(* CODESYS project osmos_MXO_added.export

Project tree, tasks and I/O mapping:
  DUT/
    data type AI_Ctr
    data type AI_Par
    data type AO_Ctr
    data type AO_Par
    data type DI_Ctr
    data type DI_Par
    data type DO_Ctr
    data type DO_Par
    data type Motor_Ctr
    data type Motor_Data
    data type Motor_Par
    data type Valve_Ctr
    data type Valve_Data
    data type Valve_Par
  FB/
    CM/
      function block CM_AI [ST]
      function block CM_AO [ST]
      function block CM_DI [ST]
      function block CM_DO [ST]
      function block CM_Motor_dozz [ST]
      function block CM_Valve_dozz [ST]
    function block CLK_1_sec [ST]
    function block _USR_CTU [ST]
  Popup/
    visualisation popup_AI
    visualisation popup_AO
    visualisation popup_DO
    visualisation popup_Motor
    visualisation popup_Sensor
    visualisation popup_Valve
*)

// DUT/AI_Ctr
TYPE AI_Ctr :
STRUCT
	ManMode:		BOOL := FALSE; //False - Auto, True - Manual
	ManValue:		REAL; 
END_STRUCT
END_TYPE

// DUT/AI_Par
TYPE AI_Par :
STRUCT
	Raw_MIN:		REAL := 0;
	Raw_MAX:		REAL := 100;
	Eng_MIN:		REAL := 0;
	Eng_MAX:		REAL := 100;
	Filter_Constant:REAL;// From 0 to 1
	Filter_Time:	UINT;//Time for filter in seconds	
END_STRUCT
END_TYPE

// DUT/AO_Ctr
TYPE AO_Ctr :
STRUCT
	ManMode:		BOOL := FALSE; //False - Auto, True - Manual
	ManValue:		REAL; 
END_STRUCT
END_TYPE

// DUT/AO_Par
TYPE AO_Par :
STRUCT	
	Eng_MIN:		REAL := 0;
	Eng_MAX:		REAL := 100;
	Raw_MIN:		REAL := 0;
	Raw_MAX:		REAL :=1000;
END_STRUCT
END_TYPE

// DUT/DI_Ctr
TYPE DI_Ctr :
STRUCT
	ManMode:		BOOL := FALSE; //False - Auto, True - Manual
	ManAct:			BOOL; 
END_STRUCT
END_TYPE

// DUT/DI_Par
TYPE DI_Par :
STRUCT
	Debounce_On:	UINT := 100; //Delay in milliseconds
	Debounce_Off:	UINT := 100; //Delay in milliseconds
END_STRUCT
END_TYPE

// DUT/DO_Ctr
TYPE DO_Ctr :
STRUCT
	ManMode:		BOOL := FALSE; //False - Auto, True - Manual
	ManAct:			BOOL; 
END_STRUCT
END_TYPE

// DUT/DO_Par
TYPE DO_Par :
STRUCT
	Debounce_On:	UINT; //Delay in milliseconds
	Debounce_Off:	UINT; //Delay in milliseconds
END_STRUCT
END_TYPE

// DUT/Motor_Ctr
TYPE Motor_Ctr :
STRUCT
	ManMode:		BOOL := FALSE; //False - Auto, True - Manual
	ManAct:			BOOL;
	AlmSuppress:	BOOL; 
END_STRUCT
END_TYPE

// DUT/Motor_Data
TYPE Motor_Data :
STRUCT
	xActivate:		BOOL;
	xFault:			BOOL;
	xOut:			BOOL;
	dwColor:		DWORD;
END_STRUCT
END_TYPE

// DUT/Motor_Par
TYPE Motor_Par :
STRUCT
	On_Delay:		UINT := 0; //all delays are set in seconds only
	Off_Delay:		UINT := 0;
	ActFlt_Delay:	UINT := 5;
	DeactFlt_Delay:	UINT := 5;
END_STRUCT
END_TYPE

// DUT/Valve_Ctr
TYPE Valve_Ctr :
STRUCT
	ManMode:		BOOL := FALSE; //False - Auto, True - Manual
	ManAct:			BOOL;
	ManActUS:		BOOL;
	ManActLS:		BOOL;
	AlmSuppress:	BOOL; 
END_STRUCT
END_TYPE

// DUT/Valve_Data
TYPE Valve_Data :
STRUCT
	xActivate:		BOOL;
	xActUpSeat:		BOOL;
	xActLowSeat:	BOOL;
	xFault:			BOOL;
	xOut:			BOOL;
	dwColor:		DWORD;
END_STRUCT
END_TYPE

// DUT/Valve_Par
TYPE Valve_Par :
STRUCT
	On_Delay:		UINT := 0; //all delays are set in seconds only
	Off_Delay:		UINT := 0;
	ActFlt_Delay:	UINT := 8;
	DeactFlt_Delay:	UINT := 8;	
END_STRUCT
END_TYPE

// FB/CLK_1_sec
FUNCTION_BLOCK CLK_1_sec
VAR_INPUT
	EN:		BOOL;
	PT:		TIME := T#1S;
END_VAR
VAR_OUTPUT
	Q:		BOOL;
END_VAR
VAR
	M:		BOOL;
	t_last:	TIME;
	tm:		TIME;
END_VAR

// This block is used for making blink-signal in a certain time with duration 1 cycle

tm := TIME();
// R_TRIG for initialization, to enable Q, when start
IF EN AND NOT M THEN
	t_last := tm - PT;  
END_IF
M := EN;

Q := tm - t_last > PT;
IF Q THEN
	t_last := tm;
END_IF

END_FUNCTION_BLOCK

// FB/_USR_CTU
FUNCTION_BLOCK _USR_CTU
VAR_INPUT
	EN:		BOOL;
	PV:		UINT;// Preset value
	CU:		BOOL;// Count input
END_VAR
VAR_OUTPUT
	Q:		BOOL;// Output
	CV:		UINT;// Current value
END_VAR
VAR	
END_VAR

// user counter up is made, to be used in ST (because in standart variant no EN/ENO)
IF NOT EN THEN
	Q := FALSE;
	CV := 0;
	RETURN;
ELSE
	IF NOT Q AND CU THEN
		CV := CV + 1;// Increase value by 1 while EN is TRUE and NOT Q
	END_IF
END_IF
Q := CV >= PV;

END_FUNCTION_BLOCK

// FB/CM/CM_AI
FUNCTION_BLOCK CM_AI
VAR_INPUT
	Name:			STRING;
	rIn:			REAL;
	Par:			AI_Par;
END_VAR
VAR_IN_OUT
	Ctrl:			AI_Ctr;
END_VAR
VAR_OUTPUT
	rOut:			REAL;
END_VAR
VAR
	xManModeMem:	BOOL;
	rOutMem:		REAL;
END_VAR
VAR_TEMP
	rOutTmp:		REAL;
END_VAR

// Scale 4..20 mA to 0..100% (for example)
rOutTmp := SCALE_R(
		IN:= rIn, 
		IN_LO:= Par.Raw_MIN, 
		IN_HI:= Par.Raw_MAX, 
		OUT_LO:= Par.Eng_MIN, 
		OUT_HI:= Par.Eng_MAX);
		
// Auto-Manual mode		
IF Ctrl.ManMode THEN
	IF NOT xManModeMem THEN // R_TRIG
		Ctrl.ManValue := rOutTmp;
	END_IF
	rOutTmp := Ctrl.ManValue; // Assign Man value in Engineering unit to Out (after scale)
END_IF
xManModeMem := Ctrl.ManMode; // Memory bit for R_TRIG Man mode

// Filter 
IF PLC_PRG.xFirstScan THEN//Initialization
	rOutMem := 0;
END_IF

IF Par.Filter_Constant < 1 AND Par.Filter_Constant > 0 AND NOT Ctrl.ManMode THEN
	rOutTmp := Par.Filter_Constant * rOutMem + (1 - Par.Filter_Constant) * rOutTmp;
END_IF

rOut := rOutMem := rOutTmp;

END_FUNCTION_BLOCK

// FB/CM/CM_AO
FUNCTION_BLOCK CM_AO
VAR_INPUT
	Name:			STRING;
	rIn:			REAL;
	Par:			AO_Par;
END_VAR
VAR_IN_OUT
	Ctrl:			AO_Ctr;
END_VAR
VAR_OUTPUT
	rOut:			REAL;
	rOutVisu:		REAL;
END_VAR
VAR
	xManModeMem:	BOOL;	
END_VAR
VAR_TEMP
	rInTmp: 		REAL;		
END_VAR

rInTmp := rIn;

// Auto-Manual mode	
IF Ctrl.ManMode THEN
	IF NOT xManModeMem THEN // R_TRIG
		Ctrl.ManValue := rInTmp;
	END_IF
	rInTmp := Ctrl.ManValue; // Assign Man value in Engineering unit to In before scale
END_IF
xManModeMem := Ctrl.ManMode; //Memory bit for R_TRIG Man mode
rOutVisu := rInTmp;
// Scale from Engineering unit to Raw value (for example: 0..100% => 4..20 mA)
rOut := SCALE_R(
		IN:= rInTmp, 
		IN_LO:= Par.Eng_MIN, 
		IN_HI:= Par.Eng_MAX, 
		OUT_LO:= Par.Raw_MIN, 
		OUT_HI:= Par.Raw_MAX);

END_FUNCTION_BLOCK

// FB/CM/CM_DI
FUNCTION_BLOCK CM_DI
VAR_INPUT
	Name:		STRING;
	xIn:		BOOL;
	Par:		DI_par;
END_VAR
VAR_IN_OUT
	Ctrl:		DI_Ctr;
END_VAR
VAR_OUTPUT
	xOut:		BOOL;
END_VAR
VAR
	xM:			BOOL;
	xManModeMem:BOOL;
	tStart:		TIME;	
END_VAR
VAR_TEMP
	tmpDebounceON:	TIME;
	tmpDebounceOFF:	TIME;
END_VAR

xOut := xIn;// Activation without filters when Parameters = 0

// Delay to activate output
IF Par.Debounce_On >0 THEN 
	tmpDebounceON := UINT_TO_TIME(Par.Debounce_On);
	IF xIn AND NOT xM THEN// R_TRIG
		tStart := TIME();
	END_IF
	xOut := xIn AND ((TIME() - tStart) > tmpDebounceON);		
END_IF

// Delay to deactivate output
IF Par.Debounce_Off >0 THEN
	tmpDebounceOFF := UINT_TO_TIME(Par.Debounce_Off);
	IF xM AND NOT xIn THEN// F_TRIG
		tStart := TIME();
	END_IF
	IF NOT xIn AND ((TIME() - tStart) < tmpDebounceOFF) THEN
		xOut := TRUE;
	END_IF		
END_IF

IF Ctrl.ManMode THEN
	IF NOT xManModeMem THEN
		Ctrl.ManAct := xOut;
	END_IF
	xOut := Ctrl.ManAct;
END_IF

xM := xIn;
xManModeMem := Ctrl.ManMode;

END_FUNCTION_BLOCK

// FB/CM/CM_DO
FUNCTION_BLOCK CM_DO
VAR_INPUT
	Name:		STRING;
	xIn:		BOOL;
	Par:		DO_par;
END_VAR
VAR_IN_OUT
	Ctrl:		DO_Ctr;
END_VAR
VAR_OUTPUT
	xOut:		BOOL;
END_VAR
VAR
	xM:			BOOL;
	xManModeMem:BOOL;
	tStart:		TIME;	
END_VAR
VAR_TEMP
	tmpDebounceON:	TIME;
	tmpDebounceOFF:	TIME;
END_VAR

xOut := xIn;// Activation without filters when Parameters = 0

// Delay to activate output
IF Par.Debounce_On >0 THEN 
	tmpDebounceON := UINT_TO_TIME(Par.Debounce_On);
	IF xIn AND NOT xM THEN// R_TRIG
		tStart := TIME();
	END_IF
	xOut := xIn AND ((TIME() - tStart) > tmpDebounceON);		
END_IF

// Delay to deactivate output
IF Par.Debounce_Off >0 THEN
	tmpDebounceOFF := UINT_TO_TIME(Par.Debounce_Off);
	IF xM AND NOT xIn THEN// F_TRIG
		tStart := TIME();
	END_IF
	IF NOT xIn AND ((TIME() - tStart) < tmpDebounceOFF) THEN
		xOut := TRUE;
	END_IF		
END_IF

IF Ctrl.ManMode THEN
	IF NOT xManModeMem THEN
		Ctrl.ManAct := xOut;
	END_IF
	xOut := Ctrl.ManAct;
END_IF

xM := xIn;
xManModeMem := Ctrl.ManMode;

END_FUNCTION_BLOCK

// FB/CM/CM_Motor_dozz
FUNCTION_BLOCK CM_Motor_dozz
VAR_INPUT
	Name:			STRING;
	Config:			BYTE;	
	FB:				BOOL;
	Rst:			BOOL;
	Motor_Par:		Motor_Par;
END_VAR
VAR_IN_OUT
	Act:			BOOL;
	Motor_Ctr:		Motor_Ctr;
END_VAR
VAR_OUTPUT
	Q:				BOOL;
	Flt:			BOOL;
END_VAR
VAR
	D_F_CTU:		_USR_CTU;
	A_F_CTU:		_USR_CTU;
	D_D_CTU:		_USR_CTU;
	A_D_CTU:		_USR_CTU;
	xAct:			BOOL;	
	xDeAct:			BOOL;
	xActDlyDone:	BOOL;
	xDeActDlyDone:	BOOL;
	Act_temp_old:	BOOL;
	ManModeMem:		BOOL;
	xGlobalAlmSupMem:	BOOL;
	dwColor:		DWORD;	
END_VAR
VAR_TEMP
	Act_temp:		BOOL;
	FB_En:			BOOL;
	RstIn_En:		BOOL;
END_VAR

Q := FALSE; 

// Read config
FB_En 		:= Config.0;
RstIn_En 	:= Config.1;

// Read parameters
A_F_CTU(PV := Motor_Par.ActFlt_Delay, CU := PLC_PRG.xCLK_1_sec);// parameters for act fault
D_F_CTU(PV := Motor_Par.DeactFlt_Delay, CU := PLC_PRG.xCLK_1_sec);// parameters for deact fault
A_D_CTU(PV := Motor_Par.On_Delay, CU:= PLC_PRG.xCLK_1_sec);// parameters for act delay
D_D_CTU(PV := Motor_Par.Off_Delay, CU:= PLC_PRG.xCLK_1_sec);// parameters for deact delay

// Reset input
IF RstIn_En THEN
	Act_temp := Act;	// Assign input to to internal variable
	Act := FALSE;
END_IF

// Auto/Man mode
IF Motor_Ctr.ManMode THEN
	IF NOT ManModeMem THEN // Detect R_trig
		Motor_Ctr.ManAct := Act_temp;		
	END_IF
	Act_temp := Motor_Ctr.ManAct;	
END_IF
ManModeMem := Motor_Ctr.ManMode;

// Activations
// Detect F_trig and R_trig activation, to SET/RESET timers
IF Act_temp AND NOT Act_temp_old THEN// R_trig activation
	xAct := TRUE;// set value on activation	
	xDeAct := FALSE;
	xActDlyDone := FALSE;
	IF NOT xDeActDlyDone THEN
		xActDlyDone := TRUE;// disable Act delay timer if DeAct delay timer is not done (Motor is activated yet)
	END_IF
	D_D_CTU.EN := FALSE;
END_IF
IF Act_temp_old AND NOT Act_temp THEN// F_trig activation
	xDeAct := TRUE;
	xAct :=FALSE;
	xDeActDlyDone := FALSE;
	IF NOT xActDlyDone THEN
		xDeActDlyDone := TRUE; // disable DeAct delay timer if Act delay timer is not done (Motor is not activated yet)
	END_IF
	A_D_CTU.EN := FALSE;
END_IF

// Activation delay
IF xAct THEN
	IF A_D_CTU.PV > 0 AND NOT xActDlyDone THEN
		A_D_CTU.EN := TRUE;//start timer 
		IF A_D_CTU.Q THEN
			xActDlyDone :=TRUE;
			A_D_CTU.EN := FALSE;
		END_IF	
	ELSE
		Q := Act_temp;
	END_IF	
END_IF
	
// Deactivation delay
IF xDeAct THEN
	IF D_D_CTU.PV > 0 AND NOT xDeActDlyDone THEN
		D_D_CTU.EN := TRUE;//Start timer
		Q := TRUE; 
		IF 	D_D_CTU.Q THEN
			xDeActDlyDone := TRUE;
			D_D_CTU.EN := FALSE;			
		END_IF
	ELSE
		Q := Act_temp;
	END_IF
END_IF


 //Activating fault timers, when Feedback is used	
IF FB_En THEN
	// Act_fault delay
	IF xAct AND Q AND NOT FB THEN
		A_F_CTU.EN :=TRUE;// Start timer 
		IF A_F_CTU.Q THEN 
			Flt := TRUE;
		END_IF
	ELSE
		A_F_CTU.EN := FALSE;
	END_IF
	// Deact fault delay
	IF xDeAct AND FB AND NOT Q THEN
		D_F_CTU.EN :=TRUE;// Start timer 
		IF D_F_CTU.Q THEN
			Flt := TRUE;
		END_IF
	ELSE
		D_F_CTU.EN :=FALSE;
	END_IF
END_IF

// Global fault reset handling
IF PLC_PRG.xGlobalAlmSup AND NOT xGlobalAlmSupMem THEN
	Motor_Ctr.AlmSuppress := TRUE;
END_IF
IF xGlobalAlmSupMem  AND NOT PLC_PRG.xGlobalAlmSup THEN
	Motor_Ctr.AlmSuppress := FALSE;
END_IF
xGlobalAlmSupMem := PLC_PRG.xGlobalAlmSup;

// Fault reset
IF Motor_Ctr.AlmSuppress OR Rst THEN
	Flt := FALSE;
END_IF

// Colors
dwColor := Const.Color_Def;

IF Q THEN
	dwColor := Const.Color_Green;
END_IF

IF Flt THEN
	dwColor := Const.Color_Fault;
END_IF

Act_temp_old := Act_temp;

END_FUNCTION_BLOCK

// FB/CM/CM_Valve_dozz
FUNCTION_BLOCK CM_Valve_dozz
VAR_INPUT
	Name:			STRING;
	Config:			BYTE;	
	FB:				BOOL;
	Rst:			BOOL;
	Act_UpperSeat:	BOOL;
	Act_LowerSeat:	BOOL;
	Valve_Par:		Valve_Par;
END_VAR
VAR_IN_OUT
	Act:			BOOL;

	Valve_Ctr:		Valve_Ctr;
END_VAR
VAR_OUTPUT
	Q:				BOOL;
	Q_UpperSeat:	BOOL;
	Q_LowerSeat:	BOOL;
	Flt:			BOOL;
	dwColor:		DWORD;
END_VAR
VAR
	D_F_CTU:		_USR_CTU;
	A_F_CTU:		_USR_CTU;
	D_D_CTU:		_USR_CTU;
	A_D_CTU:		_USR_CTU;
	xAct:			BOOL;	
	xDeAct:			BOOL;
	xActDlyDone:	BOOL;
	xDeActDlyDone:	BOOL;
	Act_temp_old:	BOOL;
	ManModeMem:		BOOL;
END_VAR
VAR_TEMP
	Act_temp:		BOOL;
	Act_US_temp:	BOOL;
	Act_LS_temp:	BOOL;
	FB_En:			BOOL;
	FB_temp:		BOOL;
	RstIn_En:		BOOL;
END_VAR

Q := Q_UpperSeat := Q_LowerSeat := FALSE; 
Act_temp := Act;// Assighn input to to internal variable

// Read config
FB_En 		:= Config.0;
RstIn_En 	:= Config.1;

FB_temp := FB;
IF Config.3 THEN // deact FB
	FB_temp := NOT FB;
END_IF

// Read parameters
A_F_CTU(PV := Valve_Par.ActFlt_Delay, CU := PLC_PRG.xCLK_1_sec);// parameters for act fault
D_F_CTU(PV := Valve_Par.DeactFlt_Delay, CU := PLC_PRG.xCLK_1_sec);// parameters for deact fault
A_D_CTU(PV := Valve_Par.On_Delay, CU:= PLC_PRG.xCLK_1_sec);// parameters for act delay
D_D_CTU(PV := Valve_Par.Off_Delay, CU:= PLC_PRG.xCLK_1_sec);// parameters for deact delay

// Seat temp act
Act_US_temp := Act_UpperSeat;
Act_LS_temp := Act_LowerSeat;

// Auto/Man mode
IF Valve_Ctr.ManMode THEN
	IF NOT ManModeMem THEN // Detect R_trig
		Valve_Ctr.ManAct := Act_temp;
		Valve_Ctr.ManActUS := Act_US_temp;
		Valve_Ctr.ManActLS := Act_LS_temp;
	END_IF
	Act_temp := Valve_Ctr.ManAct;
	Act_US_temp := Valve_Ctr.ManActUS;
	Act_LS_temp := Valve_Ctr.ManActLS;
END_IF
ManModeMem := Valve_Ctr.ManMode;

// Activations
// Detect F_trig and R_trig activation, to SET/RESET timers
IF Act_temp AND NOT Act_temp_old THEN// R_trig activation
	xAct := TRUE;// set value on activation	
	xDeAct := FALSE;
	xActDlyDone := FALSE;
	IF NOT xDeActDlyDone THEN
		xActDlyDone := TRUE;// disable Act delay timer if DeAct delay timer is not done (valve is activated yet)
	END_IF
	D_D_CTU.EN := FALSE;
END_IF
IF Act_temp_old AND NOT Act_temp THEN// F_trig activation
	xDeAct := TRUE;
	xAct :=FALSE;
	xDeActDlyDone := FALSE;
	IF NOT xActDlyDone THEN
		xDeActDlyDone := TRUE; // disable DeAct delay timer if Act delay timer is not done (valve is not activated yet)
	END_IF
	A_D_CTU.EN := FALSE;
END_IF

// Activation delay
IF xAct THEN
	IF A_D_CTU.PV > 0 AND NOT xActDlyDone THEN
		A_D_CTU.EN := TRUE;//start timer 
		IF A_D_CTU.Q THEN
			xActDlyDone :=TRUE;
			A_D_CTU.EN := FALSE;
		END_IF	
	ELSE
		Q := Act_temp;
	END_IF	
END_IF
	
// Deactivation delay
IF xDeAct THEN
	IF D_D_CTU.PV > 0 AND NOT xDeActDlyDone THEN
		D_D_CTU.EN := TRUE;//Start timer
		Q := TRUE; 
		IF 	D_D_CTU.Q THEN
			xDeActDlyDone := TRUE;
			D_D_CTU.EN := FALSE;			
		END_IF
	ELSE
		Q := Act_temp;
	END_IF
END_IF


 //Activating fault timers, when Feedback is used	
IF FB_En THEN
	// Act_fault delay
	IF xAct AND Q AND NOT FB_temp THEN
		A_F_CTU.EN :=TRUE;// Start timer 
		IF A_F_CTU.Q THEN 
			Flt := TRUE;
		END_IF
	ELSE
		A_F_CTU.EN := FALSE;
	END_IF
	// Deact fault delay
	IF xDeAct AND FB_temp AND NOT Q THEN
		D_F_CTU.EN :=TRUE;// Start timer 
		IF D_F_CTU.Q THEN
			Flt := TRUE;
		END_IF
	ELSE
		D_F_CTU.EN :=FALSE;
	END_IF
END_IF

// Global fault reset
IF PLC_PRG.xGlobalAlmSup THEN
	Valve_Ctr.AlmSuppress := TRUE;
END_IF

// Fault reset
IF Valve_Ctr.AlmSuppress OR Rst THEN
	Flt := FALSE;
END_IF

// Seat activation
IF Config.2 THEN // Mixproof valve
	Q_UpperSeat := Act_US_temp;
	Q_LowerSeat := Act_LS_temp;
END_IF

// Colors
dwColor := Const.Color_Def;

IF Q THEN
	dwColor := Const.Color_Green;
END_IF

IF Flt THEN
	dwColor := Const.Color_Fault;
END_IF

Act_temp_old := Act_temp;

END_FUNCTION_BLOCK

// Popup/popup_AI
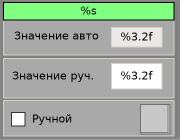
VISUALIZATION popup_AI  // 180x140
VAR_INPUT
	AICfg: 	POINTER TO CM_AI;
	AICtrl:	POINTER TO AI_Ctr;
END_VAR
    Rectangle (0,0 180x138)
        OnMouseClick: execute { SensorVis:=2; }
    Rectangle (3,2 171x53)
    Rectangle (3,2 171x18), "%s", text variable: AICfg^.Name
    Rectangle (3,100 171x36)
    Button (140,104 30x30), image: ImagePool.exit
        OnMouseClick:  Dialog=popup_AI, Result=OK, NumpadKeypadSet=True
    Rectangle (3,58 171x40)
    Label (9,61 95x30), "Значение руч."
    Checkbox (9,107 110x24), "Ручной", variable: AICtrl^.ManMode
    Textfield (111,63 51x26), "%3.2f", text variable: AICtrl^.ManValue, input disabled if: not AICtrl^.ManMode
        OnMouseClick: write the text variable via VisuDialogs.Numpad, min 0, max 100
    Label (11,21 95x30), "Значение авто"
    Textfield (111,27 51x20), "%3.2f", text variable: AICfg^.rOut
    hotkey  Id=481037385728, Key=KeyDown=True, KeyName=ESCAPE, VisuElemId=31
    hotkey  Id=481038434304, Key=KeyName=ESCAPE, VisuElemId=31
END_VISUALIZATION

// Popup/popup_AO
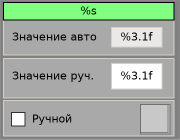
VISUALIZATION popup_AO  // 180x140
VAR_INPUT
	AOCfg: 	POINTER TO CM_AO;
	AOCtrl:	POINTER TO AO_Ctr;
END_VAR
    Rectangle (0,0 180x138)
        OnMouseClick: execute { SensorVis:=2; }
    Rectangle (3,2 171x53)
    Rectangle (3,2 171x18), "%s", text variable: AOCfg^.Name
    Rectangle (3,100 171x36)
    Button (140,104 30x30), image: ImagePool.exit
        OnMouseClick:  Dialog=popup_AO, Result=OK, NumpadKeypadSet=True
    Rectangle (3,58 171x40)
    Label (9,61 95x30), "Значение руч."
    Checkbox (9,107 110x24), "Ручной", variable: AOCtrl^.ManMode
    Textfield (111,63 51x26), "%3.1f", text variable: AOCtrl^.ManValue, input disabled if: not AOCtrl^.ManMode
        OnMouseClick: write the text variable via VisuDialogs.Numpad, min 0, max 100
    Label (9,22 95x30), "Значение авто"
    Textfield (111,27 51x20), "%3.1f", text variable: AOCfg^.rIn
    hotkey  Id=481037385728, Key=KeyDown=True, KeyName=ESCAPE, VisuElemId=31
    hotkey  Id=481038434304, Key=KeyName=ESCAPE, VisuElemId=31
END_VISUALIZATION

// Popup/popup_DO
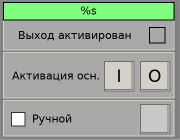
VISUALIZATION popup_DO  // 180x140
VAR_INPUT
	QCfg: 	POINTER TO CM_DO;
	QCtrl:	POINTER TO DO_Ctr;
END_VAR
    Rectangle (0,0 180x138)
        OnMouseClick: execute { SensorVis:=2; }
    Rectangle (3,2 171x48)
    Rectangle (3,2 171x18), "%s", text variable: QCfg^.Name
    Rectangle (3,100 171x36)
    Button (140,104 30x30), image: ImagePool.exit
        OnMouseClick:  Dialog=popup_DO, Result=OK, NumpadKeypadSet=True
    Rectangle (3,52 171x46)
    Label (9,61 95x30), "Активация осн."
    Rectangle (149,27 16x16), colour toggle: QCfg^.xOut
    Label (12,25 126x21), "Выход активирован"
    Checkbox (9,107 110x24), "Ручной", variable: QCtrl^.ManMode
    Button (104,61 30x30), "I", colour toggle: QCfg^.xOut, input disabled if: not QCtrl^.ManMode
        OnMouseClick: execute { QCtrl^.ManAct := TRUE; }
    Button (140,61 30x30), "O", colour toggle: not QCfg^.xOut, input disabled if: not QCtrl^.ManMode
        OnMouseClick: execute { QCtrl^.ManAct := FALSE; }
    hotkey  Id=481037385728, Key=KeyDown=True, KeyName=ESCAPE, VisuElemId=31
    hotkey  Id=481038434304, Key=KeyName=ESCAPE, VisuElemId=31
END_VISUALIZATION

// Popup/popup_Motor
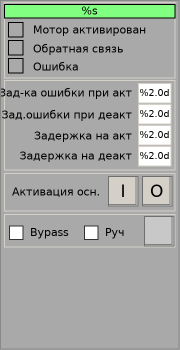
VISUALIZATION popup_Motor  // 180x350
//{attribute 'var_in_out_as_pointer'}
VAR_INPUT 
	M_Cfg: 	POINTER TO CM_Motor_dozz;
	M_Cmd:	POINTER TO Motor_Ctr;
	M_Par:	POINTER TO Motor_Par;
END_VAR
    Rectangle (4,80 171x90)
    Rectangle (4,2 171x76)
    Rectangle (4,4 171x14), "%s", text variable: M_Cfg^.Name
    Rectangle (4,214 171x33)
    Textfield (138,83 33x20), "%2.0d", text variable: M_Par^.ActFlt_Delay
        OnMouseClick: write the text variable via VisuDialogs.Numpad, min 0, max 99
    Label (6,78 129x30), "Зад-ка ошибки при акт"
    Textfield (138,104 33x20), "%2.0d", text variable: M_Par^.DeactFlt_Delay
        OnMouseClick: write the text variable via VisuDialogs.Numpad, min 0, max 99
    Label (6,100 129x30), "Зад.ошибки при деакт"
    Textfield (138,125 33x20), "%2.0d", text variable: M_Par^.On_Delay
        OnMouseClick: write the text variable via VisuDialogs.Numpad, min 0, max 30
    Label (7,121 128x30), "Задержка на акт"
    Textfield (138,146 33x20), "%2.0d", text variable: M_Par^.Off_Delay
        OnMouseClick: write the text variable via VisuDialogs.Numpad, min 0, max 30
    Label (7,141 128x30), "Задержка на деакт"
    Rectangle (4,173 171x38)
    Button (108,176 30x30), "I", colour toggle: M_Cfg^.Q, input disabled if: not M_Cmd^.ManMode
        OnMouseClick: execute { M_Cmd^.ManAct := TRUE; }
    Button (142,176 30x30), "O", colour toggle: not M_Cfg^.Q, input disabled if: not M_Cmd^.ManMode
        OnMouseClick: execute { M_Cmd^.ManAct := FALSE; }
    Label (9,177 95x30), "Активация осн."
    Checkbox (7,219 75x27), "Bypass", variable: M_Cmd^.AlmSuppress
    Checkbox (82,219 56x27), "Руч", variable: M_Cmd^.ManMode
    Button (144,216 30x30), image: ImagePool.exit
        OnMouseClick:  Dialog=popup_Motor, Result=OK, NumpadKeypadSet=True
    Label (30,21 126x18), "Мотор активирован"
    Rectangle (8,22 15x15), colour toggle: M_Cfg^.Q
    Rectangle (8,40 15x15), colour toggle: M_Cfg^.FB
    Label (30,40 126x18), "Обратная связь"
    Rectangle (8,58 15x15), colour toggle: M_Cfg^.Flt
    Label (30,58 57x18), "Ошибка"
END_VISUALIZATION

// Popup/popup_Sensor
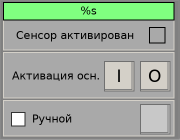
VISUALIZATION popup_Sensor  // 180x140
VAR_INPUT
	SCfg: 	POINTER TO CM_DI;
	SCtrl:	POINTER TO DI_Ctr;
END_VAR
    Rectangle (0,0 180x138)
        OnMouseClick: execute { SensorVis:=2; }
    Rectangle (3,2 171x48)
    Rectangle (3,2 171x18), "%s", text variable: SCfg^.Name
    Rectangle (3,100 171x36)
    Button (140,104 30x30), image: ImagePool.exit
        OnMouseClick:  Dialog=popup_Sensor, Result=OK, NumpadKeypadSet=True
    Rectangle (3,52 171x46)
    Label (9,61 95x30), "Активация осн."
    Rectangle (149,27 16x16), colour toggle: SCfg^.xOut
    Label (12,25 126x21), "Сенсор активирован"
    Checkbox (9,107 110x24), "Ручной", variable: SCtrl^.ManMode
    Button (104,61 30x30), "I", colour toggle: SCfg^.xOut, input disabled if: not SCtrl^.ManMode
        OnMouseClick: execute { SCtrl^.ManAct := TRUE; }
    Button (140,61 30x30), "O", colour toggle: not SCfg^.xOut, input disabled if: not SCtrl^.ManMode
        OnMouseClick: execute { SCtrl^.ManAct := FALSE; }
    hotkey  Id=481037385728, Key=KeyDown=True, KeyName=ESCAPE, VisuElemId=31
    hotkey  Id=481038434304, Key=KeyName=ESCAPE, VisuElemId=31
END_VISUALIZATION

// Popup/popup_Valve
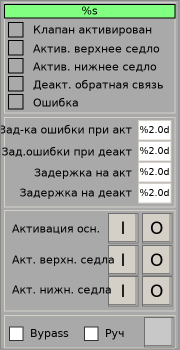
VISUALIZATION popup_Valve  // 180x350
//{attribute 'var_in_out_as_pointer'}
VAR_INPUT 
	V_Cfg: 	POINTER TO CM_Valve_dozz;
	V_Cmd:	POINTER TO Valve_Ctr;
	V_Par:	POINTER TO Valve_Par;
END_VAR
    Rectangle (4,117 171x90)
    Rectangle (4,2 171x111)
    Rectangle (4,4 171x14), "%s", text variable: V_Cfg^.Name
    Rectangle (4,315 171x33)
    Textfield (138,120 33x20), "%2.0d", text variable: V_Par^.ActFlt_Delay
        OnMouseClick: write the text variable via VisuDialogs.Numpad, min 0, max 99
    Label (6,115 129x30), "Зад-ка ошибки при акт"
    Textfield (138,141 33x20), "%2.0d", text variable: V_Par^.DeactFlt_Delay
        OnMouseClick: write the text variable via VisuDialogs.Numpad, min 0, max 99
    Label (6,137 129x30), "Зад.ошибки при деакт"
    Textfield (138,162 33x20), "%2.0d", text variable: V_Par^.On_Delay
        OnMouseClick: write the text variable via VisuDialogs.Numpad, min 0, max 30
    Label (7,158 128x30), "Задержка на акт"
    Textfield (138,183 33x20), "%2.0d", text variable: V_Par^.Off_Delay
        OnMouseClick: write the text variable via VisuDialogs.Numpad, min 0, max 30
    Label (7,178 128x30), "Задержка на деакт"
    Rectangle (4,210 171x101)
    Button (108,213 30x30), "I", colour toggle: V_Cfg^.Q, input disabled if: not V_Cmd^.ManMode
        OnMouseClick: execute { V_Cmd^.ManAct := TRUE; }
    Button (142,213 30x30), "O", colour toggle: not V_Cfg^.Q, input disabled if: not V_Cmd^.ManMode
        OnMouseClick: execute { V_Cmd^.ManAct := FALSE; }
    Button (108,245 30x30), "I", colour toggle: V_Cfg^.Q_UpperSeat, input disabled if: not V_Cmd^.ManMode
        OnMouseClick: execute { V_Cmd^.ManActUS := TRUE; }
    Button (142,245 30x30), "O", colour toggle: not V_Cfg^.Q_UpperSeat, input disabled if: not V_Cmd^.ManMode
        OnMouseClick: execute { V_Cmd^.ManActUS := FALSE; }
    Button (108,276 30x30), "I", colour toggle: V_Cfg^.Q_LowerSeat, input disabled if: not V_Cmd^.ManMode
        OnMouseClick: execute { V_Cmd^.ManActLS := TRUE; }
    Button (142,276 30x30), "O", colour toggle: not V_Cfg^.Q_LowerSeat, input disabled if: not V_Cmd^.ManMode
        OnMouseClick: execute { V_Cmd^.ManActLS := FALSE; }
    Label (9,214 95x30), "Активация осн."
    Label (9,245 103x30), "Акт. верхн. седла"
    Label (9,275 103x30), "Акт. нижн. седла"
    Checkbox (7,320 75x27), "Bypass", variable: V_Cmd^.AlmSuppress
    Checkbox (82,320 56x27), "Руч", variable: V_Cmd^.ManMode
    Button (144,317 30x30), image: ImagePool.exit
        OnMouseClick:  Dialog=popup_Valve, Result=OK, NumpadKeypadSet=True
    Label (30,21 126x18), "Клапан активирован"
    Rectangle (8,22 15x15), colour toggle: V_Cfg^.Q
    Rectangle (8,40 15x15), colour toggle: V_Cfg^.Q_UpperSeat
    Label (30,40 126x18), "Актив. верхнее седло"
    Rectangle (8,58 15x15), colour toggle: V_Cfg^.Q_LowerSeat
    Label (30,58 126x18), "Актив. нижнее седло"
    Rectangle (8,76 15x15), colour toggle: V_Cfg^.FB
    Label (30,76 126x18), "Деакт. обратная связь"
    Rectangle (8,94 15x15), colour toggle: V_Cfg^.Flt
    Label (30,94 57x18), "Ошибка"
END_VISUALIZATION
